// TwinCAT 3 PLC project HorstmanPLC
// ProgramVersion: 3.1.4023.0
// libraries:
//   Tc2_ControllerToolbox, * (Beckhoff Automation GmbH)
//   Tc2_Drive, * (Beckhoff Automation GmbH)
//   Tc2_MC2, * (Beckhoff Automation GmbH)
//   Tc2_MC2_Drive, * (Beckhoff Automation GmbH)
//   Tc2_Standard, * (Beckhoff Automation GmbH)
//   Tc2_System, * (Beckhoff Automation GmbH)
//   Tc2_Utilities, * (Beckhoff Automation GmbH)
//   Tc3_Module, * (Beckhoff Automation GmbH)
// project tree:
//   DUTs/ MoveBuffer1kms.TcDUT, Setpoint_Interface.TcDUT
//   GVLs/ Control.TcGVL, Global_Variables.TcGVL, IO.TcGVL, RecipeData.TcGVL, SAFETY.TcGVL
//   / PlcTask.TcTTO
//   POUs/FB/ FB_UseExtSetpointGen.TcPOU
//   POUs/ FB_SinGen.TcPOU, FB_ChirpGen.TcPOU, FB_TcJoy.TcPOU (not stored), MAIN.TcPOU, P_FaultMonitoring.TcPOU, P_FunctionGenerators.TcPOU, P_HMI_Polling.TcPOU, P_MotorControl.TcPOU, p_MotorControl_ST.TcPOU, P_sinGenerator.TcPOU, p_TextModeRead.TcPOU
// real-time tasks:
//   TASK PlcTask: cycle T#10ms, priority 20, ADS port 350
// motion (NC):
//   TASK NC-Task 1 SAF: cycle T#2ms, priority 4, ADS port 501
//   TASK NC-Task 1 SVB: cycle T#10ms, priority 8, ADS port 511
//   AXIS Axis 1 (id 1)
//     Dynamic: Acceleration=8000, Deceleration=8000, Jerk=32000
//     PositionAreaControl: Enable=false
//     TargetPosControl: Enable=false
//     OtherSettings: AllowMotionCmdToSlave=true
//     encoder EncType=19
//       EncPara: ScaleFactorNumerator=1.283836e-05, MaxCount=#xffffffff
//     drive DrvType=16
//       DrvPara: MaxCount=#xffffffff
//         Analog: TorqueSetpointScale=10, ScaleFactorActTorque=0.1
//         TimeComp: TaskDelayCycles=1
//     controller CtrType=1
//       CtrPara: PriorControlFactor=1
//         PosDiffControl: Enable=false
//         Observer: BandWidth=20
//   AXIS Axis 2 (id 2)
//     Dynamic: Acceleration=8000, Deceleration=8000, Jerk=32000
//     PositionAreaControl: Enable=false
//     TargetPosControl: Enable=false, Range=1
//     OtherSettings: AllowMotionCmdToSlave=true
//     encoder EncType=19
//       EncPara: ScaleFactorNumerator=1.283836e-05, MaxCount=#xffffffff
//     drive DrvType=16
//       DrvPara: MaxCount=#xffffffff
//         Analog: TorqueSetpointScale=10, ScaleFactorActTorque=0.1
//         TimeComp: TaskDelayCycles=1
//     controller CtrType=1
//       CtrPara: PriorControlFactor=1
//         PosDiffControl: Enable=false
//         Observer: BandWidth=20
//   AXIS AbsEncoders (id 3)
//     OtherSettings: AllowMotionCmdToSlave=true
//     encoder EncType=5
//       EncPara: Offset=-30.087, ReferenceSystem=1
//     drive DrvType=5
//       Analog: TorqueSetpointScale=10, ScaleFactorActTorque=0.1
//     controller CtrType=1
//       CtrPara: PriorControlFactor=1
//         Observer: BandWidth=20
//   AXIS AbsEncoders_2 (id 4)
//     OtherSettings: AllowMotionCmdToSlave=true
//     encoder EncType=5
//       EncPara: Offset=-1.4684, ReferenceSystem=1
//     drive DrvType=5
//       Analog: TorqueSetpointScale=10, ScaleFactorActTorque=0.1
//     controller CtrType=1
//       CtrPara: PriorControlFactor=1
//         Observer: BandWidth=20
// I/O:
//   DEVICE Device 1 (EtherCAT) (disabled), AmsNetId 5.63.228.160.2.1
//   DEVICE PLC IO CARDS (EtherCAT), AmsNetId 10.0.75.1.4.1
//     PLC IO (EK1200) [EK1200-5000 EtherCAT Power supply (2A E-Bus)]
//       Digital In (EL1004) [EL1004 4Ch. Dig. Input 24V, 3ms]
//       Digital Out (EL2004) [EL2004 4Ch. Dig. Output 24V, 0.5A]
//       Analog In (EL3102) [EL3102 2Ch. Ana. Input +/-10V, Diff.]
//       Analog Out (EL4032) [EL4032 2Ch. Ana. Output +/-10V, 12bit]
//       Linear Encoders [EL5002 2Ch. SSI Encoder]
//       Lasers (EL6224) [EL6224 (IO Link Master)]
//       Load Cell 12v Power (EL9512) [EL9512 Power supply terminal 12V]
//       Load Cell 1 (EL3356) -SN213902 [EL3356 1Ch. Ana. Input Resistor Bridge Terminal, 16bit, High Precision]
//       Load Cell 2 (EL3356) -sn 213903 [EL3356 1Ch. Ana. Input Resistor Bridge Terminal, 16bit, High Precision]
//       Term 20 (EL9011) [EL9011 End Terminal]
//   DEVICE Device 7 (CX5140-0121-M510) (disabled), AmsNetId 10.0.75.1.8.1
//   DEVICE Device 4 (EtherCAT Automation Protocol) (disabled), AmsNetId 192.168.0.1.5.1
//   DEVICE Drives (EtherCAT), AmsNetId 192.168.0.1.9.1
//     Drive 1 (AKD) [AKD EtherCAT Drive (CoE)]
//     Drive 2 (AKD) [AKD EtherCAT Drive (CoE)]
//   DEVICE Device 9 (COM Port) (disabled)
// variable links:
//   NC-Task 1 SAF/Axes/AbsEncoders <-> PLC IO CARDS (EtherCAT)/PLC IO (EK1200)/Linear Encoders
//     Enc/Inputs/In/nDataIn1 <-> SSI Inputs Channel 1/Counter value
//     Enc/Inputs/In/nState1 <-> SSI Inputs Channel 1/Status/Data error
//     Enc/Inputs/In/nState1 @bit 3 <-> SSI Inputs Channel 1/Status/Data mismatch
//     Enc/Inputs/In/nState1 @bit 1 <-> SSI Inputs Channel 1/Status/Frame error
//     Enc/Inputs/In/nState1 @bit 2 <-> SSI Inputs Channel 1/Status/Power failure
//     Enc/Inputs/In/nState2 @bit 5 <-> SSI Inputs Channel 1/Status/Sync error
//     Enc/Inputs/In/nState2 @bit 6 <-> SSI Inputs Channel 1/Status/TxPDO State
//     Enc/Inputs/In/nState2 @bit 7 <-> SSI Inputs Channel 1/Status/TxPDO Toggle
//     Enc/Inputs/In/nState4 @bit 1 <-> WcState/InputToggle
//     Enc/Inputs/In/nState4 <-> WcState/WcState
//   NC-Task 1 SAF/Axes/AbsEncoders_2 <-> PLC IO CARDS (EtherCAT)/PLC IO (EK1200)/Linear Encoders
//     Enc/Inputs/In/nDataIn1 <-> SSI Inputs Channel 2/Counter value
//     Enc/Inputs/In/nState1 <-> SSI Inputs Channel 2/Status/Data error
//     Enc/Inputs/In/nState1 @bit 3 <-> SSI Inputs Channel 2/Status/Data mismatch
//     Enc/Inputs/In/nState1 @bit 1 <-> SSI Inputs Channel 2/Status/Frame error
//     Enc/Inputs/In/nState1 @bit 2 <-> SSI Inputs Channel 2/Status/Power failure
//     Enc/Inputs/In/nState2 @bit 5 <-> SSI Inputs Channel 2/Status/Sync error
//     Enc/Inputs/In/nState2 @bit 6 <-> SSI Inputs Channel 2/Status/TxPDO State
//     Enc/Inputs/In/nState2 @bit 7 <-> SSI Inputs Channel 2/Status/TxPDO Toggle
//     Enc/Inputs/In/nState4 @bit 1 <-> WcState/InputToggle
//     Enc/Inputs/In/nState4 <-> WcState/WcState
//   NC-Task 1 SAF/Axes/Axis 1 <-> Drives (EtherCAT)/Drive 1 (AKD)
//     Drive/Inputs/In/nDcOutputTime <-> InfoData/DcOutputShift
//     Drive/Inputs/In/nState1 <-> TPDO mapping parameter 258/Statusword
//     Drive/Inputs/In/nState2 <-> TPDO mapping parameter 258/Statusword @bit 8
//     Drive/Inputs/In/nState4 @bit 1 <-> WcState/InputToggle
//     Drive/Inputs/In/nState4 <-> WcState/WcState
//     Drive/Outputs/Out/nCtrl1 <-> RPDO mapping parameter 258/Controlword
//     Drive/Outputs/Out/nCtrl2 <-> RPDO mapping parameter 258/Controlword @bit 8
//     Drive/Outputs/Out/nDataOut1 <-> RPDO mapping parameter 258/1st set-point
//     Enc/Inputs/In/nDataIn1 <-> TPDO mapping parameter 258/Position actual internal value
//     Enc/Inputs/In/nDcInputTime <-> InfoData/DcInputShift
//     Enc/Inputs/In/nState4 @bit 1 <-> WcState/InputToggle
//     Enc/Inputs/In/nState4 <-> WcState/WcState
//   NC-Task 1 SAF/Axes/Axis 2 <-> Drives (EtherCAT)/Drive 2 (AKD)
//     Drive/Inputs/In/nDcOutputTime <-> InfoData/DcOutputShift
//     Drive/Inputs/In/nState1 <-> TPDO mapping parameter 258/Statusword
//     Drive/Inputs/In/nState2 <-> TPDO mapping parameter 258/Statusword @bit 8
//     Drive/Inputs/In/nState4 @bit 1 <-> WcState/InputToggle
//     Drive/Inputs/In/nState4 <-> WcState/WcState
//     Drive/Outputs/Out/nCtrl1 <-> RPDO mapping parameter 258/Controlword
//     Drive/Outputs/Out/nCtrl2 <-> RPDO mapping parameter 258/Controlword @bit 8
//     Drive/Outputs/Out/nDataOut1 <-> RPDO mapping parameter 258/1st set-point
//     Enc/Inputs/In/nDataIn1 <-> TPDO mapping parameter 258/Position actual internal value
//     Enc/Inputs/In/nDcInputTime <-> InfoData/DcInputShift
//     Enc/Inputs/In/nState4 @bit 1 <-> WcState/InputToggle
//     Enc/Inputs/In/nState4 <-> WcState/WcState
//   HorstmanPLC/HorstmanPLC Instance <-> Device 1 (EtherCAT)
//     PlcTask Inputs/IO.devstate <-> Inputs/DevState
//   HorstmanPLC/HorstmanPLC Instance <-> PLC IO CARDS (EtherCAT)/PLC IO (EK1200)/Digital Out (EL2004)
//     PlcTask Outputs/IO.DriveEnable1 <-> Channel 1/Enable Drive 1
//     PlcTask Outputs/IO.DriveEnable2 <-> Channel 3/Enable Drive 2
//   HorstmanPLC/HorstmanPLC Instance <-> PLC IO CARDS (EtherCAT)/PLC IO (EK1200)/Lasers (EL6224)
//     PlcTask Inputs/IO.LaserDistanceValue <-> IO-Link Port1/Distance
//   HorstmanPLC/HorstmanPLC Instance <-> PLC IO CARDS (EtherCAT)/PLC IO (EK1200)/Load Cell 1 (EL3356) -SN213902
//     PlcTask Inputs/IO.LoadCell1 <-> RMB Value (INT32)/IO.LoadCell1
//   HorstmanPLC/HorstmanPLC Instance <-> PLC IO CARDS (EtherCAT)/PLC IO (EK1200)/Load Cell 2 (EL3356) -sn 213903
//     PlcTask Inputs/IO.LoadCell2 <-> RMB Value (INT32)/IO.LoadCell2
//   HorstmanPLC/HorstmanPLC Instance <-> NC-Task 1 SAF/Axes/Axis 1
//     PlcTask Inputs/IO.DriveAxis1.NcToPlc <-> Outputs/ToPlc
//     PlcTask Outputs/IO.DriveAxis1.PlcToNc <-> Inputs/FromPlc
//   HorstmanPLC/HorstmanPLC Instance <-> NC-Task 1 SAF/Axes/Axis 2
//     PlcTask Inputs/IO.DriveAxis2.NcToPlc <-> Outputs/ToPlc
//     PlcTask Outputs/IO.DriveAxis2.PlcToNc <-> Inputs/FromPlc

CONFIGURATION HorstmanPLC
    RESOURCE PLC ON TwinCAT3
        TASK PlcTask(INTERVAL := T#10ms, PRIORITY := 20);
        PROGRAM MAIN WITH PlcTask : MAIN;
    END_RESOURCE
END_CONFIGURATION

// ---- DUTs/MoveBuffer1kms.TcDUT
TYPE MoveBuffer1kms :
STRUCT
block:	ARRAY[0..1000] OF LREAL;
END_STRUCT
END_TYPE

// ---- DUTs/Setpoint_Interface.TcDUT

TYPE Setpoint_interface :
STRUCT
	Position :LREAL; //used by external setpoint gen blocks.
	Velocity :LREAL; //used by external setpoint gen blocks.
	Acceleration:LREAL; //used by external setpoint gen blocks. 
	Direction :DINT; //used by external setpoint gen blocks. (STOP 0, FWD 1, REV -1)
END_STRUCT
END_TYPE

// ---- GVLs/Control.TcGVL
{attribute 'qualified_only'}
VAR_GLOBAL
b_UseExternalSetpointGenerator :BOOL; // Allows fine control of servos.
b_HaltRequest: BOOL;// System is performing a halt
b_HaltRequestExecute: BOOL; //activates the halt functions
n_ServosHalted :usint; // each servo will set a 1 here in it's respective bit when halted
b_Servos_Halted :BOOL; // if all servos are in halt state, we can drop enable.
b_EnableServosFinal :BOOL; // if true, the servos will try to enable
b_SetpointGeneratorFault: BOOL;
n_RowsReadfromCsv : UDINT;
n_LastReadCSVRow :LREAL;
b_RequestCSVRead :BOOL;
sp_ServoB: Setpoint_Interface;
sp_ServoA: Setpoint_Interface;
	b_EnableServosReq: BOOL;
	b_RequestServoReset: BOOL;
	bExecMoveRelA: BOOL;
	b_ExecuteGearIn: BOOL;
	RequestedMoveVelocity : LREAL := 50;
	bAbsMoveAExecute: BOOL;
	fTargetPosA: LREAL;
	fTargetPosB: LREAL;
	fTargetVelA: LREAL;
	bAbsMoveBExecute: BOOL;
	bPlayCsv: Bool;
	fTargetVelB: LREAL;
	nPlayBackIndex: UDINT;
	RequestedState: INT;
	bAbsoluteJog: BOOL;
	bAbsoluteMoveExec: BOOL;
	bRelativeJog: BOOL;
	bRelativeMoveExec: BOOL;
END_VAR

// ---- GVLs/Global_Variables.TcGVL
{attribute 'qualified_only'}
VAR_GLOBAL
	TcJoy : FB_TcJoy;
	HmiButtonData0 : DINT;
	HmiButtonData1  : DINT;
	HmiBoolDword0 : DINT;
	HmiBoolDword1 : DINT;
	EnablemsClock: BOOL;
	msClockValid: BOOL;
	
	HMI_Servo1_Pos : LREAL;
	//HMI_Servo1_Torque : LREAL;
	HMI_Servo1_Vel : LREAL;
	HMI_Servo1_Force AT %I* :LREAL;
	
	HMI_Servo2_Pos : LREAL;
	//HMI_Servo2_Torque : LREAL;
	HMI_Servo2_Vel : LREAL;
	HMI_Servo2_Force AT %I* :LREAL;
	
	ReqVelocity :LREAL; // How fast to execute manaual action.
	ReqAccel :LREAL; // accel/decel for manual action
	Position :LREAL; // Position for manual action
	Amplitude :LREAL; // amplitude for sin function
	

	
	b_GearIn: BOOL;
	SinPeriod: TIME;
	ReqVel: TIME;
END_VAR

// ---- GVLs/IO.TcGVL
{attribute 'qualified_only'}
VAR_GLOBAL
devstate AT %I*: UINT;
SaferyOK :BOOL; // safety system status
PowerEnabled :BOOL; // soft  bit we turn on to enable drives when we have no errors.

//Outputs
//Drive 1	
TorqueRequest1 AT %Q*: INT;
DriveEnable1 AT %Q*: BOOL;
//Drive1FaultReset AT %Q*: BOOL;
DriveAxis1 : AXIS_Ref;
//Drive 2
TorqueRequest2 AT %Q*: INT;
DriveEnable2 AT %Q*:BOOL;
//Drive2FaultReset AT %Q*: BOOL;
DriveAxis2 : AXIS_Ref;


Wcstate_bus2 AT%I* :BOOL;
//Simdrive1: AXIS_Ref;
//Simdrive2: AXIS_Ref;

//Inputs
LaserDistanceValue AT %I* :UINT; // Laser
Laser2 AT %I*: UINT;
//Drive 1


Drive1digitalinBtyes  AT %I*: ARRAY[0..3] OF BYTE;
Drive1positivelimitSw: BOOL;
Drive1NegativelimitSw : BOOL;
//DriveFaulted1  AT %I*: BOOL;
//DriveEnabled1  AT %I*: BOOL;
DriveFeedback1   AT %I*: INT;
LinearPosition1   AT %I*: DINT;
LoadCell1   AT %I*: DINT;

//Drive 2
Drive2digitalinBtyes  AT %I*: ARRAY[0..3] OF BYTE;
Drive2positivelimitSw: BOOL;
Drive2NegativelimitSw : BOOL;
//DriveFaulted2  AT %I*: BOOL;
//DriveEnabled2  AT %I*: BOOL;
DriveFeedback2   AT %I*: INT;
LinearPosition2   AT %I*: DINT;
LoadCell2   AT %I*: DINT;
 
Laser_mm: LREAL;
	Encoder_Left AT %I*: UDINT;
	Encoder_Right AT %I*: UDINT;

END_VAR

// ---- GVLs/RecipeData.TcGVL
{attribute 'qualified_only'}
VAR_GLOBAL
	recipememory: ARRAY [0..1800] OF moveBuffer1kms;
END_VAR

// ---- GVLs/SAFETY.TcGVL
{attribute 'qualified_only'}
VAR_GLOBAL
	GLOBAL_SAFETY_NOT_OK: BOOL;
END_VAR

// ---- POUs/MAIN.TcPOU
PROGRAM MAIN
VAR
	SoftClock : RTC_EX;
	Chirp :fb_chirpgen;
	outputval: LREAL;
END_VAR

.Global_Variables.TcJoy(); // Read HMI data
 // read drive limit input swtich status
 io.Drive1positivelimitSw := io.Drive1digitalinBtyes[2].4;
 io.Drive1NegativelimitSw := io.Drive1digitalinBtyes[2].5;
 io.Drive2positivelimitSw := io.Drive2digitalinBtyes[2].4;
 io.Drive2NegativelimitSw := io.Drive2digitalinBtyes[2].5;
P_HMI_polling();
IF .Global_Variables.TcJoy.bIsActive THEN // if HMI is connected
	;
END_IF
p_singenerator();

chirp(en := TRUE, Reset :=FALSE, Offset := 10.0, A := 15, w1 := 10, w2 := 25,M :=2000, SignalOut => outputval);


p_FaultMonitoring(); // Check fault routine
//inputs
p_TextModeRead();
//Seq
//Outputs
P_FunctionGenerators();

SoftClock(En := Global_Variables.EnablemsClock,PMSEK:=0, Q=> Global_Variables.msClockValid);// Call for a 1ms resolution software timer to start at 0ms when enable goes true.
p_MotorControl_ST();
p_MotorControl();

//logging
//recipe system

END_PROGRAM

// ---- POUs/FB_ChirpGen.TcPOU
FUNCTION_BLOCK FB_ChirpGen
VAR_INPUT
	EN :BOOL;
	Offset: LREAL; // where to center the chirp wave in the stroke
	StartVel :LREAL;
	EndVel :LREAL;
	A :LREAL;
	M :LREAL;
	fTIME :LREAL;
	
END_VAR
VAR_OUTPUT
	SignalOut :LREAL;
END_VAR
VAR

	RESULT: LREAL;
END_VAR

Result := A * COS (startvel * ftime + (endvel - startvel) * ftime * ftime / (2*M));
signalout := result;

END_FUNCTION_BLOCK

// ---- POUs/P_HMI_Polling.TcPOU
PROGRAM P_HMI_Polling
VAR

END_VAR


Global_variables.HMI_Servo1_Pos := io.DriveAxis1.NcToPlc.ActPos;
Global_variables.HMI_Servo1_Vel := io.DriveAxis1.NcToPlc.ActVelo;
Global_variables.HMI_Servo1_force := io.LoadCell1;

Global_variables.HMI_Servo2_Pos := io.DriveAxis2.NcToPlc.ActPos;
Global_variables.HMI_Servo2_Vel := io.DriveAxis1.NcToPlc.ActVelo;
Global_variables.HMI_Servo2_force := io.LoadCell2;



Control.b_RequestServoReset := Global_variables.HmiButtonData0.3; // also passes fault reset to servo code, might want to move this to the fault monitoring routine later?

p_Faultmonitoring.b_FaultReset := Global_variables.HmiButtonData0.3; //pass fault reset to fault monitoring routine.
IF NOT p_TextmodeRead.bRead AND Global_variables.HmiButtonData0.5 THEN
control.b_RequestCSVRead :=   TRUE; 
ELSE
	control.b_RequestCSVRead :=   FALSE;
END_IF
IO.Laser_mm := UINT_TO_LREAL(io.LaserDistanceValue)  / 10.0;


IF Global_variables.HmiButtonData0.10 	THEN Control.RequestedState := 0; END_IF // Abs move mode
IF Global_variables.HmiButtonData0.11 	THEN Control.RequestedState := 1; END_IF // Rel Move Mode
IF Global_variables.HmiButtonData0.12 	THEN Control.RequestedState := 2; END_IF // Sin mode
IF Global_variables.HmiButtonData0.13 	THEN Control.RequestedState := 3; END_IF // Chirp Mode
IF Global_variables.HmiButtonData0.14 	THEN Control.RequestedState := 4; END_IF // CSV playback mode
IF Global_variables.HmiButtonData0.15 	THEN Control.RequestedState := 5; END_IF // Zeroing Mode
IF Global_variables.HmiButtonData0.16 	THEN Control.RequestedState := 6; END_IF // Jog to limits mode

 //Global_variables.HmiButtonData0.6 is execute button 



Global_variables.HmiBoolDword0.0 := io.DriveAxis1.NcToPlc.StateDWord.0; // drive 1 enable nc status
//Global_variables.HmiBoolDword0.1 := io.DriveFaulted1;
Global_variables.HmiBoolDword0.2 := io.DriveAxis2.NcToPlc.StateDWord.0; // drive 2 enable nc status
//Global_variables.HmiBoolDword0.3 := io.DriveFaulted2;
Global_variables.HmiBoolDword0.4 := Global_variables.b_GearIn;
Global_variables.HmiBoolDword0.5 := control.b_Servos_Halted;
Global_variables.HmiBoolDword0.6 := control.b_EnableServosFinal;
Global_variables.HmiBoolDword0.7 := p_Faultmonitoring.b_Faulted;

END_PROGRAM

// ---- POUs/P_FaultMonitoring.TcPOU
PROGRAM P_FaultMonitoring
VAR_INPUT
		b_FaultReset: BOOL;
		b_bool: bool;
END_VAR


VAR

	n_Fault: ARRAY [0..1] OF DINT;
	b_FaultPending :BOOL;
	b_Faulted: BOOL;
	GlobalFaultTimer: ton; // all faults are checked in this interval.
	GlobalFaultTime: TIME:= T#1S;
	SR_0: SR;

	b_FaultImmediately: BOOL;
	st_StateDwordDrive1 :NCTOPLC_AXIS_REF_STATE;
	st_StateDwordDrive2 : NCTOPLC_AXIS_REF_STATE;
END_VAR
VAR // added by the converter: edge detectors and wires of the graphical bodies
    _rt1 : R_TRIG;
    _w1 : BOOL;
END_VAR

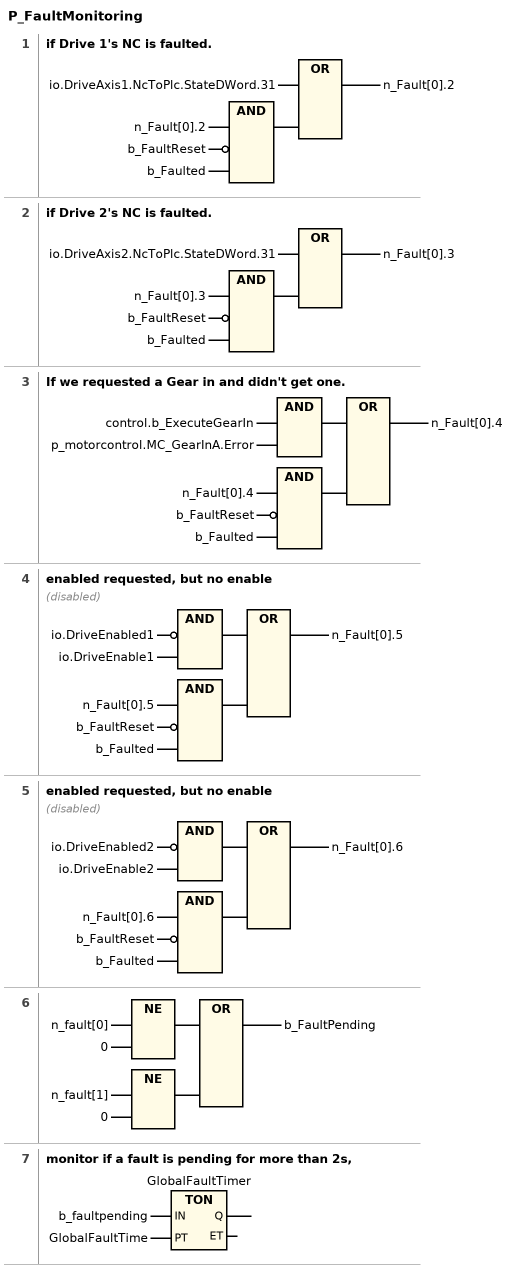
// NETWORK 1: if Drive 1's NC is faulted.
n_Fault[0].2 := io.DriveAxis1.NcToPlc.StateDWord.31 OR n_Fault[0].2 AND NOT b_FaultReset AND b_Faulted;

// NETWORK 2: if Drive 2's NC is faulted.
n_Fault[0].3 := io.DriveAxis2.NcToPlc.StateDWord.31 OR n_Fault[0].3 AND NOT b_FaultReset AND b_Faulted;

// NETWORK 3: If we requested a Gear in and didn't get one.
n_Fault[0].4 := control.b_ExecuteGearIn AND p_motorcontrol.MC_GearInA.Error OR n_Fault[0].4 AND NOT b_FaultReset AND b_Faulted;

// NETWORK 4: enabled requested, but no enable (disabled)
// n_Fault[0].5 := NOT io.DriveEnabled1 AND io.DriveEnable1 OR n_Fault[0].5 AND NOT b_FaultReset AND b_Faulted;

// NETWORK 5: enabled requested, but no enable (disabled)
// n_Fault[0].6 := NOT io.DriveEnabled2 AND io.DriveEnable2 OR n_Fault[0].6 AND NOT b_FaultReset AND b_Faulted;

// NETWORK 6
b_FaultPending := n_fault[0] <> 0 OR n_fault[1] <> 0;

// NETWORK 7: monitor if a fault is pending for more than 2s,
GlobalFaultTimer(IN := b_faultpending, PT := GlobalFaultTime); // TON

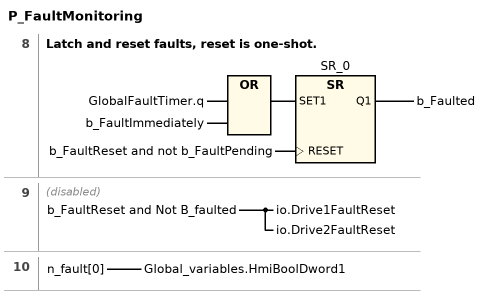
// NETWORK 8: Latch and reset faults, reset is one-shot.
_rt1(CLK := b_FaultReset and not b_FaultPending);
SR_0(SET1 := GlobalFaultTimer.q OR b_FaultImmediately, RESET := _rt1.Q); // SR
b_Faulted := SR_0.Q1;

// NETWORK 9 (disabled)
// _w1 := b_FaultReset and Not B_faulted;
// io.Drive1FaultReset := _w1;
// io.Drive2FaultReset := _w1;

// NETWORK 10
Global_variables.HmiBoolDword1 := n_fault[0];

END_PROGRAM

// ---- POUs/P_MotorControl.TcPOU
PROGRAM P_MotorControl
VAR
	
  	error:BOOL;
    fJogVelocity :LREAL;
	MC_Halt_ServoB: MC_Halt;
	MC_Halt_ServoA: MC_Halt;
	sinGen : FB_singen;	
	ServoA_SPGen: FB_useExtSetpointGen;
	ServoB_SPGen: FB_useExtSetpointGen;
	nSawSPError : INT :=0;
	r_trig_0: r_trig;


	
	b_ExecuteGearIn: BOOL;
	MC_GearInA: MC_GearIn;
	MC_MoveRelativeA: MC_MoveRelative;
	bAbsMoveBExecute: BOOL;
	MC_MoveAbsolute_A: MC_MoveContinuousAbsolute;
	ZeroingReqRtrig: R_TRIG;
	bSetZero: BOOL;
	McWritePArams1: MC_WriteParameterPersistent;
	McWritePArams2: MC_WriteParameterPersistent;
	MC_SetPosition_0: MC_SetPosition;
	MC_SetPosition_1: MC_SetPosition;
	MC_MoveAbsolute_Jog: MC_MoveAbsolute;
	MC_MoveContinuousRelative_0: MC_MoveContinuousRelative;
	MC_MoveRelative_Jog: MC_MoveRelative;
	RelMoveDistance: LREAL;
	bSinGenEnable: BOOL;
	RS_0: rs;
END_VAR
VAR // added by the converter: edge detectors and wires of the graphical bodies
    _rt1 : R_TRIG;
END_VAR

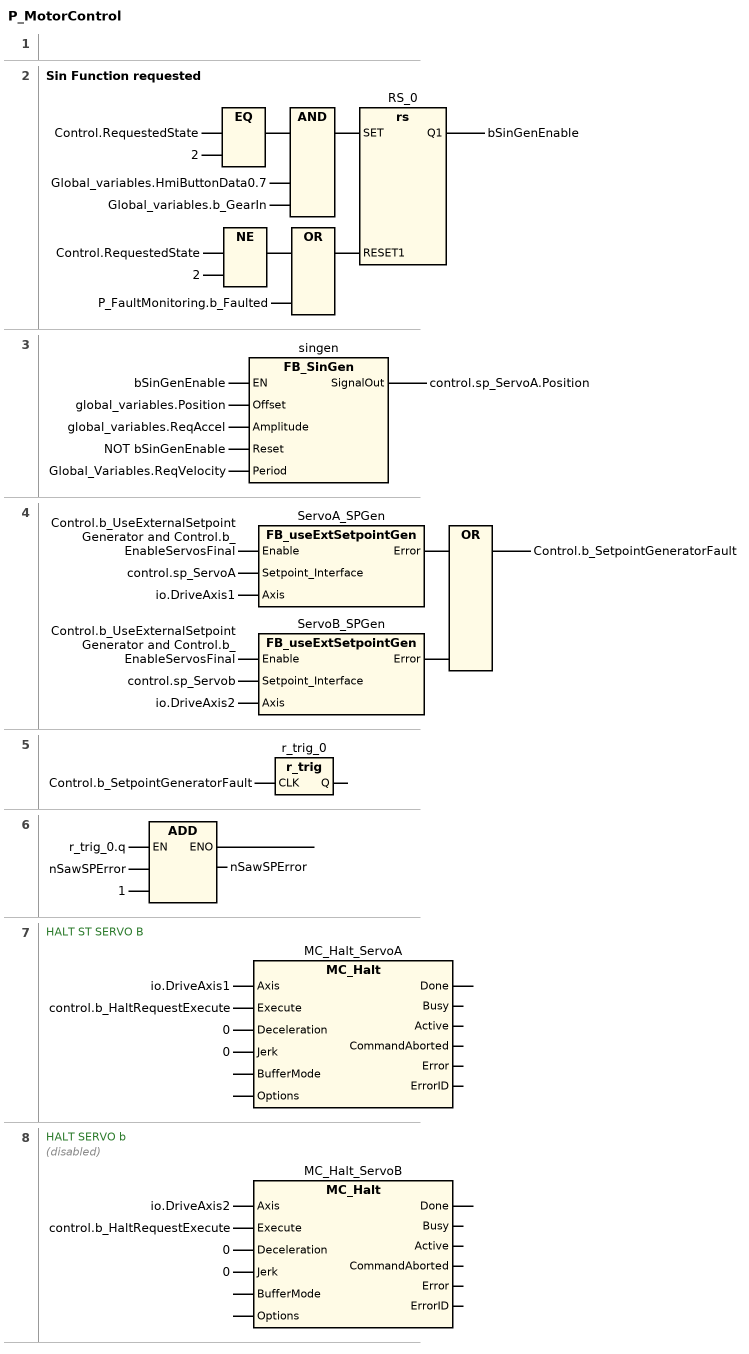
// NETWORK 1

// NETWORK 2: Sin Function requested
RS_0(SET := Control.RequestedState = 2 AND Global_variables.HmiButtonData0.7 AND Global_variables.b_GearIn, RESET1 := Control.RequestedState <> 2 OR P_FaultMonitoring.b_Faulted); // rs
bSinGenEnable := RS_0.Q1;

// NETWORK 3
singen(
    EN := bSinGenEnable,
    Offset := global_variables.Position,
    Amplitude := global_variables.ReqAccel,
    Reset := NOT bSinGenEnable,
    Period := Global_Variables.ReqVelocity); // FB_SinGen
control.sp_ServoA.Position := singen.SignalOut;

// NETWORK 4
ServoA_SPGen(
    Enable := Control.b_UseExternalSetpointGenerator and Control.b_EnableServosFinal,
    Setpoint_Interface := control.sp_ServoA,
    Axis := io.DriveAxis1); // FB_useExtSetpointGen
ServoB_SPGen(
    Enable := Control.b_UseExternalSetpointGenerator and Control.b_EnableServosFinal,
    Setpoint_Interface := control.sp_Servob,
    Axis := io.DriveAxis2); // FB_useExtSetpointGen
Control.b_SetpointGeneratorFault := ServoA_SPGen.Error OR ServoB_SPGen.Error;

// NETWORK 5
r_trig_0(CLK := Control.b_SetpointGeneratorFault); // r_trig

// NETWORK 6
IF r_trig_0.q THEN nSawSPError := nSawSPError + 1; END_IF

// NETWORK 7
// HALT ST SERVO B
MC_Halt_ServoA(Axis := io.DriveAxis1, Execute := control.b_HaltRequestExecute, Deceleration := 0, Jerk := 0); // MC_Halt

// NETWORK 8 (disabled)
// HALT SERVO b
// MC_Halt_ServoB(Axis := io.DriveAxis2, Execute := control.b_HaltRequestExecute, Deceleration := 0, Jerk := 0); // MC_Halt

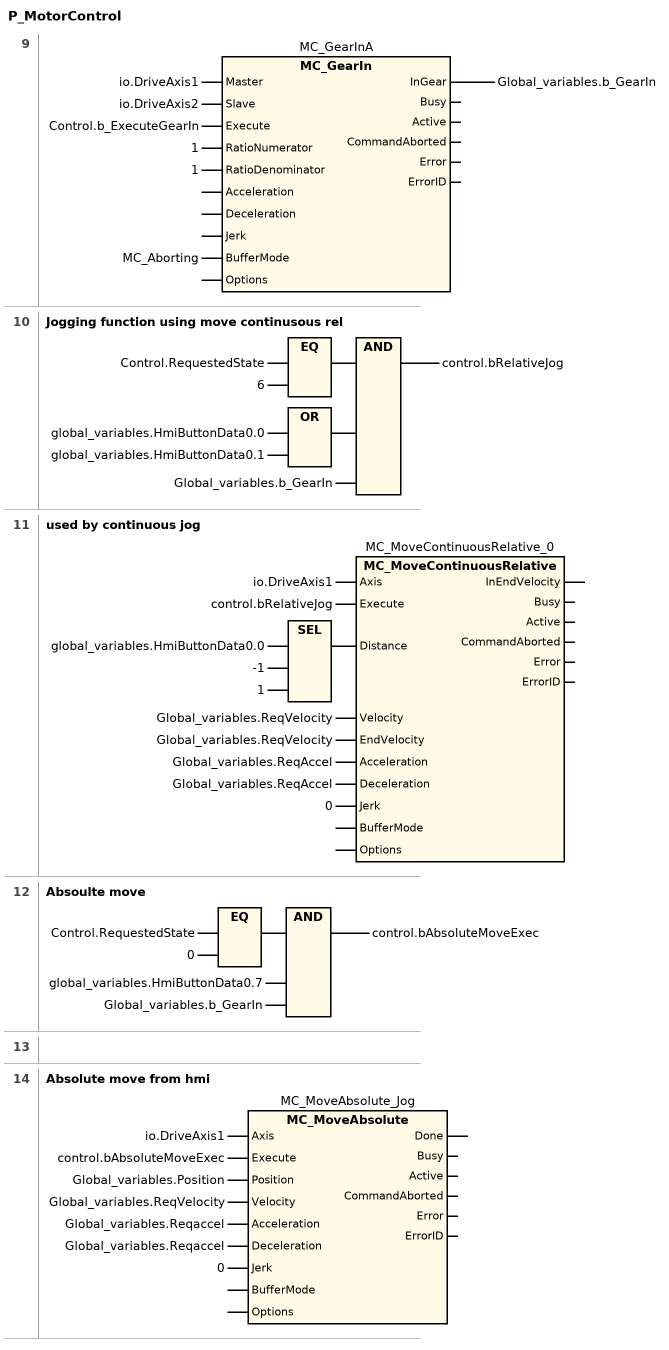
// NETWORK 9
MC_GearInA(
    Master := io.DriveAxis1,
    Slave := io.DriveAxis2,
    Execute := Control.b_ExecuteGearIn,
    RatioNumerator := 1,
    RatioDenominator := 1,
    BufferMode := MC_Aborting); // MC_GearIn
Global_variables.b_GearIn := MC_GearInA.InGear;

// NETWORK 10: Jogging function using move continusous rel
control.bRelativeJog := Control.RequestedState = 6 AND (global_variables.HmiButtonData0.0 OR global_variables.HmiButtonData0.1) AND Global_variables.b_GearIn;

// NETWORK 11: used by continuous jog
MC_MoveContinuousRelative_0(
    Axis := io.DriveAxis1,
    Execute := control.bRelativeJog,
    Distance := SEL(global_variables.HmiButtonData0.0, -1, 1),
    Velocity := Global_variables.ReqVelocity,
    EndVelocity := Global_variables.ReqVelocity,
    Acceleration := Global_variables.ReqAccel,
    Deceleration := Global_variables.ReqAccel,
    Jerk := 0); // MC_MoveContinuousRelative

// NETWORK 12: Absoulte move
control.bAbsoluteMoveExec := Control.RequestedState = 0 AND global_variables.HmiButtonData0.7 AND Global_variables.b_GearIn;

// NETWORK 13

// NETWORK 14: Absolute move from hmi
MC_MoveAbsolute_Jog(
    Axis := io.DriveAxis1,
    Execute := control.bAbsoluteMoveExec,
    Position := Global_variables.Position,
    Velocity := Global_variables.ReqVelocity,
    Acceleration := Global_variables.Reqaccel,
    Deceleration := Global_variables.Reqaccel,
    Jerk := 0); // MC_MoveAbsolute

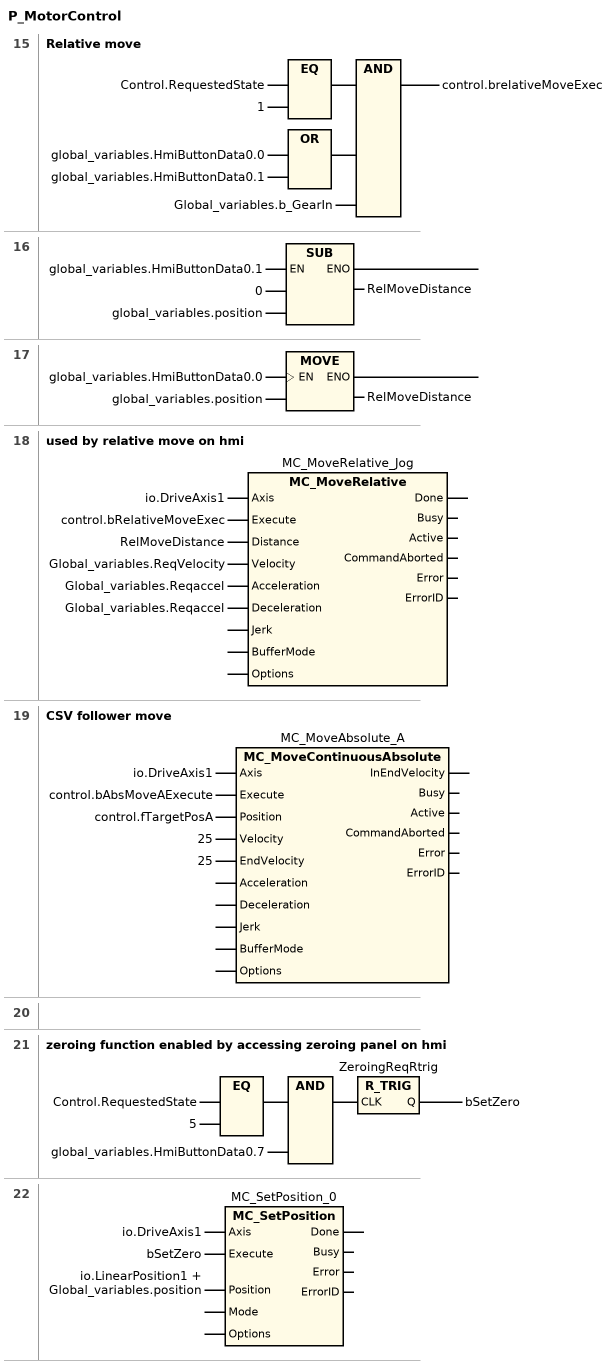
// NETWORK 15: Relative move
control.brelativeMoveExec := Control.RequestedState = 1 AND (global_variables.HmiButtonData0.0 OR global_variables.HmiButtonData0.1) AND Global_variables.b_GearIn;

// NETWORK 16
IF global_variables.HmiButtonData0.1 THEN RelMoveDistance := 0 - global_variables.position; END_IF

// NETWORK 17
_rt1(CLK := global_variables.HmiButtonData0.0);
IF _rt1.Q THEN RelMoveDistance := global_variables.position; END_IF

// NETWORK 18: used by relative move on hmi
MC_MoveRelative_Jog(
    Axis := io.DriveAxis1,
    Execute := control.bRelativeMoveExec,
    Distance := RelMoveDistance,
    Velocity := Global_variables.ReqVelocity,
    Acceleration := Global_variables.Reqaccel,
    Deceleration := Global_variables.Reqaccel); // MC_MoveRelative

// NETWORK 19: CSV follower move
MC_MoveAbsolute_A(
    Axis := io.DriveAxis1,
    Execute := control.bAbsMoveAExecute,
    Position := control.fTargetPosA,
    Velocity := 25,
    EndVelocity := 25); // MC_MoveContinuousAbsolute

// NETWORK 20

// NETWORK 21: zeroing function enabled by accessing zeroing panel on hmi
ZeroingReqRtrig(CLK := Control.RequestedState = 5 AND global_variables.HmiButtonData0.7); // R_TRIG
bSetZero := ZeroingReqRtrig.Q;

// NETWORK 22
MC_SetPosition_0(
    Axis := io.DriveAxis1,
    Execute := bSetZero,
    Position := io.LinearPosition1 + Global_variables.position); // MC_SetPosition

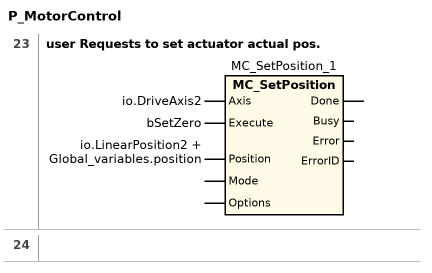
// NETWORK 23: user Requests to set actuator actual pos.
MC_SetPosition_1(
    Axis := io.DriveAxis2,
    Execute := bSetZero,
    Position := io.LinearPosition2 + Global_variables.position); // MC_SetPosition

// NETWORK 24

END_PROGRAM

// ---- POUs/FB_SinGen.TcPOU
FUNCTION_BLOCK FB_SinGen
VAR_INPUT
	EN :BOOL;
	Offset: LREAL; // where to center the sin wave in the stroke
	Amplitude :LREAL; // how much to multiply the -1 to +1 sin signal by to get the target setpoint
	Reset: BOOL;
	Period : LREAL;
END_VAR
VAR_OUTPUT
	SignalOut :LREAL;
END_VAR
VAR
	TimerPreset: TIME; // freqeuncy of sin depends on this
	K: LREAL;
	N: DINT;
	b_init: BOOL;
	RESULT: LREAL;
	Timer: TON;
	
END_VAR

IF EN THEN
	IF Reset THEN
	b_init := FALSE;
	timer.pt := LREAL_TO_TIME(period);
END_IF

IF NOT b_init THEN
    K :=2*PI/1000; (* DO ONCE *) 
	b_init := TRUE;
END_IF
timer.PT := TimerPreset;
Timer(IN := NOT timer.q);

IF timer.Q AND b_init THEN	// don't step unless initialized
N := N+1; (* REPEAT THIS *)
N :=  N MOD 1000; 
RESULT := SIN(K*N); // feeds out a sin signal from -1 to +1, scale and offset to get appropriate motion profile.
Signalout := ((Result * amplitude) + Global_variables.Position);
END_IF;
ELSE 
	Signalout := 0;
END_IF

END_FUNCTION_BLOCK

// ---- POUs/FB/FB_UseExtSetpointGen.TcPOU
FUNCTION_BLOCK FB_UseExtSetpointGen

VAR_INPUT
	Enable :BOOL; // allows motion commands, turn off to disable servo and engage brakes. don't do this while moving unless you don't want to control the decelleration ramp.
	Setpoint_Interface : Setpoint_Interface; // takes values in from the SP gen
END_VAR

VAR
	MC_ExternalSetpointGenEnable :MC_ExtSetPointGenEnable;
	MC_ExternalSetpointGenDisable :MC_ExtSetPointGenDisable;
	ErrorId: UDINT;
END_VAR

VAR_OUTPUT
	Error: BOOL;
	Enabled: BOOL;
	Busy: BOOL;
END_VAR

VAR_IN_OUT
Axis: AXIS_REF; // axis to manipulate	
END_VAR

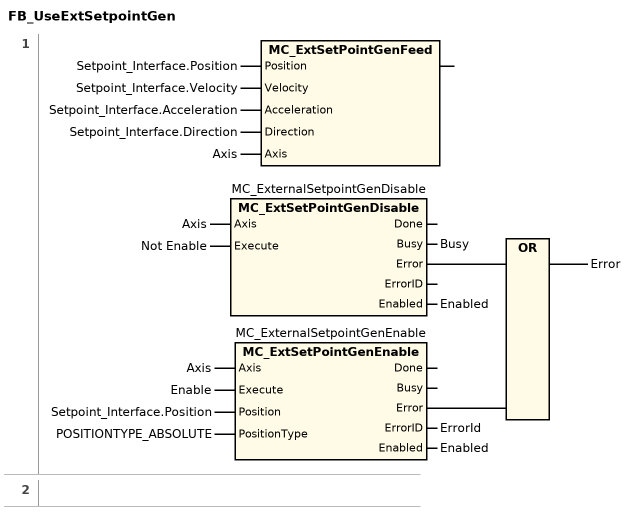
// NETWORK 1
MC_ExtSetPointGenFeed(Position := Setpoint_Interface.Position, Velocity := Setpoint_Interface.Velocity, Acceleration := Setpoint_Interface.Acceleration, Direction := Setpoint_Interface.Direction, Axis := Axis);
MC_ExternalSetpointGenDisable(Axis := Axis, Execute := Not Enable, Busy => Busy, Enabled => Enabled); // MC_ExtSetPointGenDisable
MC_ExternalSetpointGenEnable(
    Axis := Axis,
    Execute := Enable,
    Position := Setpoint_Interface.Position,
    PositionType := POSITIONTYPE_ABSOLUTE,
    ErrorID => ErrorId,
    Enabled => Enabled); // MC_ExtSetPointGenEnable
Error := MC_ExternalSetpointGenDisable.Error OR MC_ExternalSetpointGenEnable.Error;

// NETWORK 2

END_FUNCTION_BLOCK

// ---- POUs/p_TextModeRead.TcPOU
PROGRAM p_TextModeRead

VAR
	bRead			: BOOL := FALSE;(* Rising edge starts program execution *)
	sNetId			: T_AmsNetId := '';	(* TwinCAT system network address *)
	sFileName	: T_MaxString := 'C:\Twincat\FtpRoot\file.csv';(* CSV source file path and name *)
	sCSVLine		: T_MaxString := '';(* Single CSV text line (row, record), we are using string as record buffer (your are able to see read fields)  *)
	sCSVField		: T_MaxString := '';(* Single CSV field value (column, record field) *)
	bBusy			: BOOL;
	bError			: BOOL;
	nErrId			: UDINT;
	nRow	 		: UDINT 	:= 0;(* Row number (record) *)
	nColumn		: UDINT 	:= 0;(* Column number (record field) *)
	hFile			: UINT		:= 0;(* File handle of the source file *)
	step			: DWORD 	:= 0;
	fbFileOpen	: FB_FileOpen;(* Opens file *)
	fbFileClose	: FB_FileClose;(* Closes file *)
	fbFileGets		: FB_FileGets;(* Reads one record (line) *)
	fbReader		: FB_CSVMemBufferReader;(* Helper function block used to parse CSV data bytes (single record line) *)

	database		: ARRAY[0..1000] OF STRING(64);(* Target PLC database *)
	IndexList : ARRAY [0..1000] OF INT;
	
	b_initialized: BOOL;
	i: INT;
END_VAR

IF NOT b_initialized THEN
	FOR i := 0 TO 1000 DO
		
		indexlist[i] := i;
	END_FOR
	b_initialized := TRUE;
END_IF

bRead := control.b_RequestCSVRead;

CASE step OF
	0:	(* Wait for rising edge at bRead variable *)
		IF bRead THEN
			bRead 	:= FALSE;
			bBusy 		:= TRUE;
			bError		:= FALSE;
			nErrId		:= 0;
			hFile		:= 0;
			nRow	 	:= 0;
			nColumn	:= 0;
			MEMSET( ADR( database ), 0, SIZEOF( database ) );
			step 		:= 1;
		END_IF

	1:	(* Open source file *)
		fbFileOpen(  bExecute := FALSE  );
		fbFileOpen( 	sNetId := sNetId, sPathName := sFileName, nMode := FOPEN_MODEREAD OR FOPEN_MODETEXT,(* Open file in TEXT mode! *)
						ePath := PATH_GENERIC, bExecute := TRUE );
		step := 2;

	2:(* Wait until open not busy *)
		fbFileOpen( bExecute := FALSE, bError => bError, nErrID => nErrID, hFile => hFile );
		IF NOT fbFileOpen.bBusy THEN
			IF NOT fbFileOpen.bError THEN
				step := 3;
			ELSE(* Error: file not found? *)
				step := 100;
			END_IF
		END_IF

	3:	(* Read single line (record) *)
		fbFileGets( bExecute := FALSE );
		fbFileGets( sNetId := sNetId, hFile := hFile, bExecute := TRUE );
		step := 4;

	4:(* Wait until read not busy *)
		fbFileGets( bExecute := FALSE, bError => bError, nErrID => nErrID, sLine => sCSVLine );
		IF NOT fbFileGets.bBusy THEN
			IF NOT fbFileGets.bError THEN
				IF fbFileGets.bEOF THEN
					step := 10;(* End of file reached => Close source file *)
				ELSE

					(* FB_FileGets returns text line without the CR (carriage return) character.
					We have to restore the CR character (replace the $L character with $R$L characters) *)
					IF RIGHT( sCSVLine, 1 ) = '$L' THEN
						sCSVLine := REPLACE( sCSVLine, '$R$L', 2, LEN( sCSVLine ) );
					END_IF

					step := 5;
				END_IF
			ELSE(* Error *)
				step := 100;
			END_IF
		END_IF

	5:(* Parse single line (record) *)
		fbReader.eCmd := eEnumCmd_First;(* Read first field value *)
		REPEAT
			fbReader( pBuffer := ADR( sCSVLine ), cbBuffer := SIZEOF( sCSVLine ), getValue =>sCSVField );
			IF fbReader.bOk THEN
				fbReader.eCmd := eEnumCmd_Next;(* Read next field value *)

				IF ( nRow <= 1000 ) THEN
					
						database[nRow] := CSVFIELD_TO_STRING( sCSVField, FALSE );(* TODO: Save or use the field value in your application *)
					Control.n_LastReadCSVRow := STRING_TO_LREAL(database[nRow]);
				END_IF

				nColumn := nColumn + 1;(* Increment number of read columns *)
				IF fbReader.bCRLF THEN(* CRLF == TRUE => End of reacord reached *)
					nRow 		:= nRow + 1;(* Increment number of read records *)
					nColumn 	:= 0;(* Reset number of columns *)
				END_IF
control.n_RowsReadfromCsv := nrow;
			ELSE(* Error: End of record reached or all fields read *)
				step := 3;(* Try to read next line *)
			END_IF
		UNTIL NOT fbReader.bOk
		END_REPEAT

	10:	(* Close source file *)
		fbFileClose( bExecute := FALSE );
		fbFileClose( sNetId := sNetId, hFile := hFile, bExecute := TRUE );
		step := 11;

	11:(* Wait until close not busy *)
		fbFileClose( bExecute := FALSE, bError => bError, nErrID => nErrID );
		IF ( NOT fbFileClose.bBusy ) THEN
			hFile := 0;
			step := 100;
		END_IF

	100: (* Error or ready step => cleanup *)
		IF ( hFile <> 0 ) THEN
			step := 10; (* Close the source file *)
		ELSE
			bBusy := FALSE;
			step := 0;	(* Ready *)
		END_IF

END_CASE

END_PROGRAM

// ---- POUs/P_sinGenerator.TcPOU
PROGRAM P_sinGenerator
VAR
		K: LREAL;
	N: DINT;
	b_init: BOOL;
	RESULT: LREAL;
	Timer: TON;
END_VAR

IF NOT b_init THEN
    K :=2*PI/1000; (* DO ONCE *) 
	b_init := TRUE;
END_IF
timer.PT := T#10MS;
Timer(IN := NOT timer.q);

IF timer.Q THEN	
N := N+1; (* REPEAT THIS *)

N :=  N MOD 1000; 
RESULT := SIN(K*N); // feeds out a sin signal from -1 to +1, scale and offset to get appropriate motion profile.
END_IF;

END_PROGRAM

// ---- POUs/P_FunctionGenerators.TcPOU
PROGRAM P_FunctionGenerators
VAR
	
nPositionAr: ARRAY [0..2, 0..999]  OF LREAL; ///1000 positions to fill 1 second, 3 seconds worth of buffer. position data in ms.
timer: TON; //track time
ElapsedTIME :TIME;
nPostionTarget: LREAL;
nCase: INT;
SignalGenerator : FB_CTRL_SIGNAL_GENERATOR;

//sin gen
sin_bufferspace :LREAL; //10mm
sin_Magnitude : LREAL; //100 mm
sin_frequency :LREAL; // 5 hz?
sin_time :TIME;
	sin_index: lreal;
	sinout: LREAL;
	sin_steps: LREAL;
	sin_speed: LREAL;
	nSinStep: INT;
	//mc_moveAbs1: MC_moveabsolute;
	//mc_moveAbs2: MC_moveabsolute;
		mc_moveAbs1:Mc_MoveContinuousAbsolute;
	mc_moveAbs2:Mc_MoveContinuousAbsolute;
		mc_AbsCont1 :Mc_MoveContinuousAbsolute;
	haltServo1: MC_Halt;
	Runtimer: BOOL;
	bMove1 :BOOL;
	bMove2 :BOOL;
	bHalt: BOOL;
	mcabscont1buffermode : MC_buffermode := MC_blendingHigh;
	mc_movere1: MC_moveRelative;
	brelMove1: BOOL;
	relmove1Dist: LREAL;
	mc_movere2: MC_moveRelative;
	rel_speed: LREAL;
	livePosition: LREAL;
	LiveVel: LREAL := 1000;
	bMoveit: BOOL;
	n_i: INT;
	n_max: INT;
	initialized: BOOL;
	InitialPosition: LREAL;
	SignalGeneratorParams: ST_CTRL_SIGNAL_GENERATOR_PARAMS;
	SignalGenratorOutput: LREAL;
	
	SignalGeneratorErrorID: Tc2_ControllerToolbox.E_CTRL_ERRORCODES;
	SignalGeneratorError: BOOL;
	SignalType : Tc2_ControllerToolbox.E_CTRL_SIGNAL_TYPE; //  eCTRL_TRIANGLE := 0,  eCTRL_SINUS := 1,  eCTRL_SAWTOOTH := 2
	bInit: BOOL :=TRUE;
	tempvar: INT;
	PositionBuffer: LREAL;
	SignalGeneratorMode: Tc2_ControllerToolbox.E_CTRL_MODE;
	SignalGeneratorState: Tc2_ControllerToolbox.E_CTRL_STATE;
END_VAR

// these calls only run when the exectute bit is set, but must always be callable, so they go here. might need to put these at the end of this block to avoid a 1 cycle delay.
//mc_moveAbs1(Axis := io.DriveAxis1, Execute := bMove1, Position := 0, Velocity := sin_speed);
//mc_movere1(Axis := io.DriveAxis1, Execute := brelMove1, Distance:=relmove1Dist,  Velocity := rel_speed);
//mc_movere2(Axis := io.DriveAxis1, Execute := brelMove1, Distance:=relmove1Dist,  Velocity := rel_speed);
//mc_moveAbs2(Axis := io.DriveAxis1, Execute := bmove2, Position := sin_magnitude, Velocity := sin_speed);
//haltServo1(axis := io.DriveAxis1, execute := bHalt);
//mc_AbsCont1(axis := io.DriveAxis1,Position := PositionBuffer ,Velocity:= LiveVel,Execute:= bMoveit,BufferMode:=mcabscont1buffermode);
timer(in:= runtimer);
	IF bInit THEN
	(* init the setpoint array *)
	SignalGeneratorParams.tCtrlCycleTime		:= T#1MS;
	SignalGeneratorParams.tTaskCycleTime		:= T#1MS;
	SignalGeneratorParams.eSignalType			:= eCTRL_SINUS;
	SignalGeneratorParams.tStart				:= T#0mS;
	SignalGeneratorParams.tCylceDuration		:= T#100MS;
	SignalGeneratorParams.fAmplitude			:= 40;
	SignalGeneratorParams.fOffset				:= SignalGeneratorParams.fAmplitude + 10;

	(* set the mode to ACTIVE --> normal operation *)
	SignalGeneratorMode := eCTRL_MODE_ACTIVE;
	tempvar := nCase;
	(* reset init flag *)
	bInit := FALSE;
	END_IF
SignalGenerator(fManValue := InitialPosition, eMode := SignalGeneratorMode, fOut => SignalGenratorOutput, eState => SignalGeneratorState, eErrorid => SignalGeneratorErrorID, bError => SignalGeneratorError, stParams := SignalGeneratorParams);
liveposition := SignalGenratorOutput;

CASE nCase OF
	0:
	runtimer := FALSE;
	sin_index := 0;
//bInit := TRUE;	
	SignalGeneratorMode := eCTRL_MODE_RESET;
	bMoveit := FALSE;
	
	1:
	//osscillate between two positions for a period of time. not actually sin
	sin_magnitude := 100;
	sin_Frequency := 1; // hz
	sin_time := T#10S;
	Sin_index := sin_index * PI;

	sin_speed := sin_magnitude * (sin_frequency);   
   // determine velocity required for move, put it into absolute request, fire, when it gets there, fire another one to 0.
   // move 100, 200mm/s
   //move done, send next move immediately, flip flop until done.
   timer.PT := sin_time;
   timer.IN := runtimer;
   
   IF timer.Q THEN nsinstep := 4;
	
   END_IF
   CASE nSinStep OF 
	   0: //mcabsolute to 0
	   
	   IF NOT mc_moveabs1.Busy AND NOT mc_moveabs1.Error AND NOT mc_moveabs1.InEndVelocity THEN 
	   Runtimer := TRUE;	   
	   bMove1 := TRUE;
	   nSinStep := 1;
	   END_IF
	   	   1:
		   
	   IF mc_moveabs1.InEndVelocity THEN nSinstep := 2; END_IF 
		bMove1 := FALSE;
	   2:
	    
	   IF NOT mc_moveabs2.Busy AND NOT mc_moveabs2.Error AND NOT mc_moveabs2.InEndVelocity THEN 
	   Runtimer := TRUE;	   
	   bMove2 := TRUE;
	   nSinStep := 3;
	   END_IF

	   3:
	      IF mc_moveabs2.InEndVelocity THEN nSinstep := 0; END_IF 
		bMove2 := FALSE; 
   
		4:  /// exit loop
		//mcabsolute to 0, then stop.
		nSinStep := 5;
		runtimer := FALSE;
		nCase := 0;
		5:
		 IF mc_moveabs1.InEndVelocity THEN nCase := 0; END_IF
		nSinstep := 0 ;
		// wait for move 4
		6: //external setpoint experiment
	
   END_CASE
//check if timer has expired
//mc absolute move to 0
//wait for 
   

	

	
	
	2:// relative follower.
	IF NOT initialized THEN 
	n_i := 0;
	n_max := 999;
	initialized := TRUE;
	END_IF
	
	
	
	mc_AbsCont1(axis := io.DriveAxis1,Position := livePosition,Velocity:= LiveVel,Execute:= bMoveit);
	n_i := n_i +1;
	//
	liveposition:= STRING_TO_LREAL(p_TextModeRead.database[n_i]);
	IF n_i = 999 THEN
		n_i := 0;
	END_IF
	3://Sin follower.

SignalGeneratorMode := eCTRL_MODE_ACTIVE;
    IF control.sp_ServoA.Position > SignalGenratorOutput THEN
		Control.sp_ServoA.Direction := 1;
	END_IF
	IF control.sp_ServoA.Position > SignalGenratorOutput THEN
		Control.sp_ServoA.Direction := 2;
	END_IF
  IF control.sp_ServoB.Position > SignalGenratorOutput THEN
		Control.sp_ServoB.Direction := 1;
	END_IF
	IF control.sp_ServoB.Position > SignalGenratorOutput THEN
		Control.sp_ServoB.Direction := 2;
	END_IF
	
	control.sp_ServoA.Position := SignalGenratorOutput;
	control.sp_ServoB.Position := SignalGenratorOutput;
	
	
	bmoveit := FALSE;
	
IF mc_AbsCont1.InEndVelocity OR NOT mc_AbsCont1.Busy THEN
		bmoveit :=TRUE;
	END_IF
IF mc_AbsCont1.Active THEN
	bmoveit := FALSE;

END_IF	

	4://
	
END_CASE

END_PROGRAM

// ---- POUs/p_MotorControl_ST.TcPOU
PROGRAM p_MotorControl_ST
VAR
	MC_GearOutDrive1 :MC_Gearout;
	Mc_ResetServoA : MC_Reset;
	Mc_ResetServoB : MC_Reset;
	FbMc_PowerServoB :MC_Power;
	FbMc_PowerServoA :MC_Power;
	

 ServoResetOK :BYTE;
 
 jogbuttontimer :ton;
 
 //Monitor the rising edge of the ecnoder position reset function.
 
ServosReady :byte; // 	
 
// ServoEnableFallingEdge: f_trig;	
 // ServoEnableRisingEdge: r_trig;	
 // SoeResetRisingEdge :r_trig;
	st_Buffermode : MC_Buffermode;
	n_Override :INT := 100;
	SoeReset :BYTE;
	
   EncodeCalibrationRequest_RisingEdge :r_trig;
	
	b_debugSetEncoders: BOOL;
	debugging_belt: BOOL;
	BufferMode: MC_Buffermode;
	BeltForceBit: BOOL;
	state: INT; // State machine current step
	b_ServosReady: BOOL;
	b_Faulted: BOOL;
	testbool: BOOL;
	ServoDisableTimeout :Ton;
	b_DEBUG_STOP: BOOL;
	b_EncoderCalibrationRequest: BOOL;
	RequestedState: INT;
	Requested: INT;
	n_JogReq: INT;
	ServoEnableRtrig : r_trig;
	PowerEnableRtrig: r_trig;
	MoveDoneRtrig: r_trig;
	ExecuteButtonRtrig: R_trig;
	JogRtrig: R_trig;
	JogUpRtrig: R_trig;;
	JogDnRtrig: R_trig;
	B_Debubool: BOOL;
END_VAR

st_buffermode := MC_Aborting; // stop between moves instead of blending? see the mc_buffermode docs
jogbuttontimer.PT := T#250MS;
b_Faulted := p_faultmonitoring.b_Faulted;
Mc_ResetServoA(Axis := io.DriveAxis1, Execute := Control.b_RequestServoReset);
Mc_ResetServoB(Axis := io.DriveAxis2, Execute := Control.b_RequestServoReset);//STb
io.DriveEnable1 := Control.b_EnableServosFinal;
io.DriveEnable2 := control.b_EnableServosFinal ;
MC_GearOutDrive1(Slave := io.DriveAxis2, Execute := NOT Control.b_ExecuteGearIn);
servoenablertrig(CLK := io.PowerEnabled) ;
IF servoenablertrig.q THEN
	control.b_EnableServosReq := TRUE;
END_IF

PowerEnableRtrig(CLK := Global_variables.HmiButtonData0.2) ; // power on off request handler.

IF PowerEnableRtrig.q  AND NOT b_faulted THEN // if we get a power on request, and we're not faulted, try turning on power. turn it off if it's already on.
	IF io.PowerEnabled THEN 
		io.PowerEnabled := FALSE;
		ELSE
		io.PowerEnabled := TRUE;
		END_IF
	END_IF

IF b_faulted THEN io.PowerEnabled := FALSE; END_IF; // drop power on fault.


IF NOT io.PowerEnabled THEN
	control.b_EnableServosReq := false;
END_IF

IF Control.b_RequestServoReset OR b_Faulted OR NOT IO.PowerEnabled THEN // if faulted, reset, or powered off Go to state 0
state :=0; //Reset state
END_IF 






CASE state OF 
	
0: //Faulted OR Not enabled, but stopped (intialize here)
//servo power off, disable all moves and halts.			
control.b_EnableServosFinal := FALSE; // servo power off
control.b_HaltRequest := FALSE; //
control.b_UseExternalSetpointGenerator := FALSE;
control.bAbsMoveAExecute := FALSE;
control.bAbsMoveBExecute := FALSE;
 control.b_ExecuteGearIn := FALSE;

IF control.b_EnableServosReq AND (NOT b_faulted  AND NOT safety.GLOBAL_SAFETY_NOT_OK) THEN
	state := 1; // Leave the faulted state when not faulted.
	//Control.b_RequestServoReset := TRUE;
END_IF
 
1: //ready to enable, but haven't been asked to.
	 // sit here until user enable is high // user can issue reset during this stage to help wake motors.
IF NOT p_FaultMonitoring.b_Faulted AND io.PowerEnabled THEN // 
	control.b_EnableServosFinal := TRUE; // Enable the servos if the servo request is on.
//	Control.b_RequestServoReset := FALSE;	
	ELSE
		control.b_EnableServosFinal := FALSE; // Enable the servos if the servo request is on.
		State := 0;
END_IF


IF b_ServosReady THEN state := 2; END_IF; // if the servos are all enabled, we can move to next state

2: // Turning on servos with NO Commands issued, so halt them. 
control.b_HaltRequest := TRUE;	
IF control.b_Servos_Halted AND RequestedState <> 0 THEN State := RequestedState; END_IF; 

IF control.b_EnableServosReq = FALSE THEN control.b_EnableServosFinal := FALSE; State:=0; END_IF 


state := 5;	// attempt Gear in 	


3: //Switch into SP mode
	;//Enabeld, turn off halts, turn on SP generator access to servos
	control.b_HaltRequest := FALSE;
	control.b_UseExternalSetpointGenerator := TRUE;

	IF control.b_SetpointGeneratorFault	THEN State:= 4; END_IF; //halt if setpoint generator gets an error.
	IF NOT b_ServosReady THEN state := 4; END_IF; // drop power to servos if any servo loses op mode
 

4: //Enable has been dropped, HALT! (No time delay)
	control.b_UseExternalSetpointGenerator := FALSE;
 
	control.b_HaltRequest := TRUE;
   IF control.b_Servos_Halted THEN State := 0; END_IF; //drop back to initial state when halted.
   IF NOT (control.b_EnableServosReq) THEN state := 0; END_IF;
   IF ServoDisableTimeout.Q THEN State := 0; END_IF;
   
   
   
 5://gear in 

 control.b_HaltRequest := FALSE;
 control.b_ExecuteGearIn := TRUE;
 IF P_Motorcontrol.MC_GearInA.InGear THEN 
;
 END_IF

	
40: // CSV follower.
	Control.fTargetPosA := STRING_TO_LREAL(p_textmoderead.database[Control.nPlayBackIndex]);

IF NOT (p_motorcontrol.MC_MoveAbsolute_A.Active) THEN
	control.bAbsMoveAExecute := TRUE;
	State := 41;
	END_IF;
 41:
 MoveDoneRTrig(CLK := p_motorcontrol.MC_MoveAbsolute_A.InEndVelocity OR io.DriveAxis1.Status.InPositionArea);
control.bAbsMoveAExecute := FALSE;
IF MoveDoneRTrig.Q THEN // index to next move if not at end of file.

	IF Control.nPlayBackIndex <= Control.n_RowsReadfromCsv THEN
	Control.nPlayBackIndex := Control.nPlayBackIndex +1;
	State := 40;
	ELSE State := 0; 	// quit.
	END_IF

END_IF


//IF p_motorcontrol.MC_MoveAbsolute_A.error THEN state := 110; END_IF



110: 
;
111: //reached end
	;
END_CASE

Servodisabletimeout.PT := T#1000MS;
Servodisabletimeout(IN:=(state = 4)); //.q is true 2 seconds after servo enable is no longer commanded
 
//Servo enable command sent rising edge	
//ServoEnableRisingedge(CLK:=control.b_EnableServosFinal);
// lost enable, start halt & shutdown procedure
//ServoEnableFallingedge(CLK:=(Control.b_MainCoreServoEnableReq AND control.b_EnableServosReq));

//Send halt command to NC (this is here for timing reasons)
Control.b_HaltRequestExecute := control.b_HaltRequest; // halt if requested, unless the servo system is disabled.  


// pack servo readdy bits into the servoready byte. if a Bit is true, the assosiated servo is ready to roll.
Servosready.0 := io.DriveAxis1.NcToPlc.StateDWord.0;
Servosready.1 := io.DriveAxis2.NcToPlc.StateDWord.0;

IF ServosReady = 3 THEN //if all servos ready set bool true
	b_ServosReady := TRUE;
	ELSE
	b_Servosready :=FALSE;
END_IF

Control.n_ServosHalted.0 := P_MotorControl.MC_Halt_ServoB.Done;
Control.n_ServosHalted.1 := P_MotorControl.MC_Halt_ServoA.Done;

//detect when everything is halted.
IF control.n_ServosHalted = 3 THEN // change back to 255 to watch pendulum and laser
	control.b_Servos_Halted :=TRUE;
	ELSE
	control.b_Servos_Halted :=FALSE;
END_IF


//a
	FbMc_PowerServoA(Enable		:= Control.b_EnableServosFinal,
			Enable_Positive	:= Control.b_EnableServosFinal ,
			Enable_Negative	:= Control.b_EnableServosFinal ,
			Override		:= n_Override ,
			BufferMode		:= st_Buffermode ,
			Axis			:= io.DriveAxis1 );

//Servo B		
	FbMc_PowerServoB(Enable		:= Control.b_EnableServosFinal,
			Enable_Positive	:= Control.b_EnableServosFinal ,
			Enable_Negative	:= Control.b_EnableServosFinal ,
			Override		:= n_Override ,
			BufferMode		:= st_Buffermode ,
			Axis			:= io.DriveAxis2 );	

			
			// when we see execute reset a bit,
			// watch rising edge for done bit blocking it with error bit?
			//set /reset bits to fill offsets byte
			//send summary

END_PROGRAM
